Fanuc KAREL source: compact_preamble.KL

PROGRAM KC00019
%NOLOCKGROUP
VAR
I:INTEGER;J:INTEGER;K:INTEGER;R:REAL;B:BOOLEAN;S : STRING[80];T : STRING[80];AI : ARRAY[8] OF INTEGER
AB : ARRAY[244] OF BYTE
F : FILE
SA : ARRAY[8] OF STRING[80]
SB : ARRAY[8] OF STRING[80]
-- UNRESOLVED DECLARATIONS (source type spelling not recovered)
-- P : TYPE_0x001F (type_u16=0x001F)
-- Q : TYPE_0x001F (type_u16=0x001F)
BEGIN
XML_GETDATA(F,I,SA,SB,S,B,J)
END KC00019
